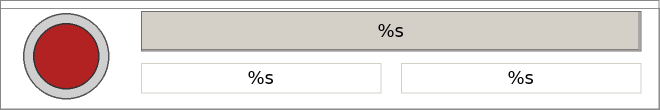
VISUALIZATION SingleDigitalOutput  // 660x110
VAR_IN_OUT
	stDigitalOutput : ST_VisuCtrlOutputFrame;
END_VAR
    GroupBox (0,0 660x110)
        Lamp1 (16,6 100x100), variable: stDigitalOutput.bOut, style: Lamp-Lamp1-Red
        Button (141,11 500x40), "%s", text variable: stDigitalOutput.sName, input disabled if: stDigitalOutput.bControlable, text list: ''
            toggle stDigitalOutput.btnOut
        Textfield (141,63 240x30), "%s", text variable: stDigitalOutput.sModuleType
        Textfield (401,63 240x30), "%s", text variable: stDigitalOutput.sPortID
END_VISUALIZATION

(* stored: Version 1.1.0.1, ProductVersion 3.1.4024.9
   Visu SingleDigitalOutput: Id {db95f671-ddfa-4ebf-861d-f4afc9969e4a} *)
